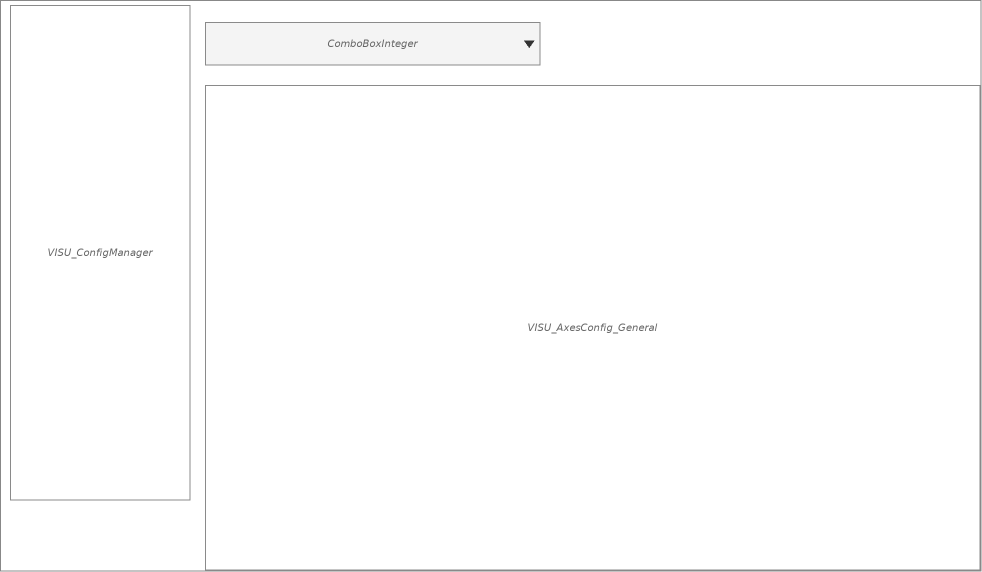
VISUALIZATION VISU_AxesConfig  // 982x572
VAR_IN_OUT
    editable : AxesConfig;
	active : AxesConfig;
    mgr : ConfigManager;
    mgrWidget : ConfigManagerWidget;
    axesWidget : AxesWidget;
END_VAR
    Frame (10,5 180x495)
        shows VISU_ConfigManager(mgr := mgr, widget := mgrWidget)
    ComboBoxInteger (205,22 335x43), variable: axesWidget.activeConfigTab, text list: 'AxesConfigTextList'
    Frame (205,85 775x485), frame switch variable: axesWidget.activeConfigTab
        shows VISU_AxesConfig_General(editable := editable, active := active)
        shows VISU_AxesConfig_KnownPositions(activePosition := axesWidget.activeConfigPosition, editable := editable.knownPositions, active := active.knownPositions)
        shows VISU_AxesConfig_Location(active := active.location, editable := editable.location)
        shows VISU_AxesConfig_LocalConditions(active := active.localConditions, editable := editable.localConditions)
        shows VISU_AxesConfig_Azimuth_1(active := active.azi, editable := editable.azi)
        shows VISU_AxesConfig_Azimuth_2(active := active.azi, editable := editable.azi)
        shows VISU_AxesConfig_Azimuth_3(active := active.azi, editable := editable.azi)
        shows VISU_AxesConfig_Elevation_1(active := active.ele, editable := editable.ele)
        shows VISU_AxesConfig_Elevation_2(active := active.ele, editable := editable.ele)
        shows VISU_AxesConfig_Rotation_1(active := active.roc, editable := editable.roc)
        shows VISU_AxesConfig_Rotation_2(active := active.roc, editable := editable.roc)
        shows VISU_AxesConfig_Rotation_1(active := active.ron, editable := editable.ron)
        shows VISU_AxesConfig_Rotation_2(active := active.ron, editable := editable.ron)
        shows VISU_AxesConfig_FilterWheel()
        shows VISU_MeasurementConfig(active := active.relativeHumidities.insideTube, editable := editable.relativeHumidities.insideTube)
        shows VISU_MeasurementConfig(active := active.dewpoints.topAir, editable := editable.dewpoints.topAir)
        shows VISU_MeasurementConfig(active := active.dewpoints.insideTube, editable := editable.dewpoints.insideTube)
        shows VISU_MeasurementConfig(active := active.accelerometers.tube.x, editable := editable.accelerometers.tube.x)
        shows VISU_MeasurementConfig(active := active.accelerometers.tube.y, editable := editable.accelerometers.tube.y)
        p1226617324: active.relativeHumidities.topAir
        p1437654724: editable.relativeHumidities.topAir
END_VISUALIZATION

(* stored: Version 1.1.0.1, ProductVersion 3.1.4019.2
   Visu VISU_AxesConfig: Id {e84c8ba7-e7cf-45fd-9359-fb9165946f43} *)
